ABB RobotStudio station: Tp3_20201123-002807.rsstn

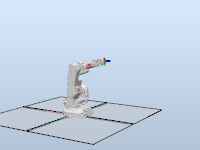
Station Tp3 (saved by RobotStudio 20.2.9116.0)
Controller IRB_140_6kg_0.81m
  mechanical unit ROB_1: IRB-140, 6 joints, base frame (0, 0, 0) mm
Layout (positions relative to the parent item):
  - IRB-140 [mechanism] at (0, 0, 0) mm; joint values [-3.0576, 0.1064, -0.4149, 0.1773, 0.2597, -2.4334] (rad or m)
      links: Base, Link1, Link2, Link3, Link4, Link5, Link6
Targets, tools, work objects and paths stored in the station, written as RAPID:
! task T_ROB1
MODULE Module1
  CONST robtarget Pos_inicial:=[[-533.014588406,-47.835810924,828.73894736],[0.635481621,-0.251423899,-0.640712069,0.349910242],[-2,0,-2,0],[9E+09,9E+09,9E+09,9E+09,9E+09,9E+09]];
  CONST robtarget BrazoAdel_CodoPos_MunNeg:=[[-533.014588406,-47.835810924,828.73894736],[0.635481621,-0.251423899,-0.640712069,0.349910242],[-2,0,-2,0],[9E+09,9E+09,9E+09,9E+09,9E+09,9E+09]];
  CONST robtarget BrazoAdel_CodoPos_MunPos:=[[-533.014588406,-47.835810924,828.73894736],[0.635481621,-0.251423899,-0.640712069,0.349910242],[-2,-2,0,1],[9E+09,9E+09,9E+09,9E+09,9E+09,9E+09]];
  CONST robtarget BrazoAdel_CodoNeg_MunNeg:=[[-533.014588406,-47.835810924,828.73894736],[0.635481621,-0.251423899,-0.640712069,0.349910242],[-2,0,-2,2],[9E+09,9E+09,9E+09,9E+09,9E+09,9E+09]];
  CONST robtarget BrazoAdel_CodoNeg_MunPos:=[[-533.014588406,-47.835810924,828.73894736],[0.635481621,-0.251423899,-0.640712069,0.349910242],[-2,-2,0,3],[9E+09,9E+09,9E+09,9E+09,9E+09,9E+09]];
  CONST robtarget BrazoAtras_CodoNeg_MunNeg:=[[-533.014588406,-47.835810924,828.73894736],[0.635481621,-0.251423899,-0.640712069,0.349910242],[0,-2,-2,4],[9E+09,9E+09,9E+09,9E+09,9E+09,9E+09]];
  CONST robtarget BrazoAtras_CodoNeg_MunPos:=[[-533.014588406,-47.835810924,828.73894736],[0.635481621,-0.251423899,-0.640712069,0.349910242],[0,0,0,5],[9E+09,9E+09,9E+09,9E+09,9E+09,9E+09]];
  CONST robtarget BrazoAtras_CodoPos_MunNeg:=[[-533.014588406,-47.835810924,828.73894736],[0.635481621,-0.251423899,-0.640712069,0.349910242],[0,-2,-2,6],[9E+09,9E+09,9E+09,9E+09,9E+09,9E+09]];
  CONST robtarget BrazoAtras_CodoPos_MunPos:=[[-533.014588406,-47.835810924,828.73894736],[0.635481621,-0.251423899,-0.640712069,0.349910242],[0,0,0,7],[9E+09,9E+09,9E+09,9E+09,9E+09,9E+09]];
  PROC Show8Configs()
    MoveJ Pos_inicial,v1000,fine,tool0\WObj:=wobj0;
    MoveJ BrazoAdel_CodoPos_MunPos,v1000,fine,tool0\WObj:=wobj0;
    MoveJ BrazoAdel_CodoPos_MunNeg,v1000,fine,tool0\WObj:=wobj0;
    MoveJ BrazoAdel_CodoNeg_MunPos,v1000,fine,tool0\WObj:=wobj0;
    MoveJ BrazoAdel_CodoNeg_MunNeg,v1000,fine,tool0\WObj:=wobj0;
    MoveJ BrazoAtras_CodoPos_MunPos,v1000,fine,tool0\WObj:=wobj0;
    MoveJ BrazoAtras_CodoPos_MunNeg,v1000,fine,tool0\WObj:=wobj0;
    MoveJ BrazoAtras_CodoNeg_MunPos,v1000,fine,tool0\WObj:=wobj0;
    MoveJ BrazoAtras_CodoNeg_MunNeg,v1000,fine,tool0\WObj:=wobj0;
    MoveJ Pos_inicial,v1000,fine,tool0\WObj:=wobj0;
  ENDPROC
  PROC main()
    Show8Configs;
  ENDPROC
ENDMODULE

